// TIA Portal V19 export
// export: Created 2026-08-08T14:07:58.6505087Z, ExportSetting WithDefaults, DisplayName Totally Integrated Automation Portal, DisplayVersion V19, DisplayName TIA Portal Openness, DisplayVersion V19, DisplayName TIA Portal Version Control Interface, DisplayVersion V19, DisplayName STEP 7 Professional, DisplayVersion V19, DisplayName STEP 7 Safety, DisplayVersion V19, DisplayName WinCC Basic/Comfort/Advanced, DisplayVersion V19, DisplayName WinCC Unified, DisplayVersion V19
ORGANIZATION_BLOCK "Main"   // OB1, LAD, ProgramCycle
TITLE = "Main Program Sweep (Cycle)"
{ S7_Optimized_Access := 'TRUE' }
VERSION : 0.1
// stored: AutoNumber true, IsIECCheckEnabled false, SetENOAutomatically false
   VAR_INPUT
      Initial_Call : Bool;
      Remanence : Bool;
   END_VAR
BEGIN

REGION Network 1
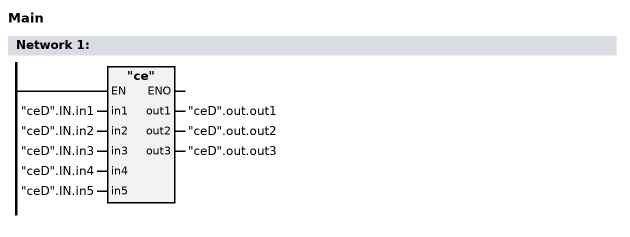
   RUNG wire#powerrail
      "ce"(in1 := "ceD".IN.in1, in2 := "ceD".IN.in2, in3 := "ceD".IN.in3, in5 := "ceD".IN.in5, in4 := "ceD".IN.in4, out1 => "ceD".out.out1, out2 => "ceD".out.out2, out3 => "ceD".out.out3)
   END_RUNG
   // the same network as SCL:
   "ce"(in1 := "ceD".IN.in1,
        in2 := "ceD".IN.in2,
        in3 := "ceD".IN.in3,
        in4 := "ceD".IN.in4,
        in5 := "ceD".IN.in5,
        out1 => "ceD".out.out1,
        out2 => "ceD".out.out2,
        out3 => "ceD".out.out3);
END_REGION
END_ORGANIZATION_BLOCK
